// TIA Portal V19 export
TYPE "C104_VAR_IF_KLP_TYPIC"
   STRUCT
      OPEN { ExternalAccessible := 'False'; ExternalVisible := 'False'; ExternalWritable := 'False'} : Bool;   // Brandstofklep open
      TOE { ExternalAccessible := 'False'; ExternalVisible := 'False'; ExternalWritable := 'False'} : Bool;   // Brandstofklep dicht
      EXT_AUT { ExternalAccessible := 'False'; ExternalVisible := 'False'; ExternalWritable := 'False'} : Bool;   // Externe (hoofd) beveiliging aangesproken
      EXT_HW { ExternalAccessible := 'False'; ExternalVisible := 'False'; ExternalWritable := 'False'} : Bool;   // Sturings hardware (PLC) in storing
      STO { ExternalAccessible := 'False'; ExternalVisible := 'False'; ExternalWritable := 'False'} : Struct   // Opsomming van alle storingen
         A001 : Bool;   // Beveiliging aangesproken
         A002 : Bool;   // Brandstofklep in storing
         A003 : Bool;   // Algemene storing brandstofklep
      END_STRUCT;
   END_STRUCT;
END_TYPE
